// TIA Portal V18 export
TYPE "LGasp_CmdAttuatori"
// stored: IsFailsafeCompliant false
   STRUCT
      attuatore : Array[1.."N_MaxAttuatoriStz"] of "LGasp_typeCmdAttuatore";
   END_STRUCT;
END_TYPE
